// TIA Portal V16 export
// export: Created 2024-06-17T18:37:11.9513972Z, ExportSetting WithDefaults, DisplayName Totally Integrated Automation Portal, DisplayVersion V16, DisplayName TIA Portal Version Control Interface, DisplayVersion V16, DisplayName TIA Portal Openness, DisplayVersion V16, DisplayName STEP 7 Professional, DisplayVersion V16, DisplayName STEP 7 Safety, DisplayVersion V16, DisplayName WinCC Advanced, DisplayVersion V16
TYPE "Axis.RB.Do_PLC.Di"
TITLE = Tabela de Entradas vindas do robô
// stored: IsFailsafeCompliant false
   STRUCT
      "RB.Go_PLC.GiPLC_NumProg" : Int;   // Retorno Número Programa em Execução
      "RB.Do_PLC.Di16_ProgramaRecebido" : Bool;   // Reconhecimento de Programa Recebido
      "RB.Do_PLC.Di17_RequisicaoPrograma" : Bool;   // Autoriza CLP a enviar Número de Programa
      "RB.Do_PLC.Di18_Home" : Bool;   // Robô em Home
      "RB.Do_PLC.Di19_FaultSumSignal" : Bool;   // Robo em Falha
      "RB.Do_PLC.Di20_SafetyChainOK" : Bool;   // Sem Falhas de Hardware nos Canais de Segurança
      "RB.Do_PLC.Di21_MotorOnState" : Bool;   // Motores Ligados
      "RB.Do_PLC.Di22_Auto_On" : Bool;   // Robô em Automático
      "RB.Do_PLC.Di23_Cycle_On" : Bool;   // Programa em Execução
      "RB.Do_PLC.Di24_EmCicloVazio" : Bool;   // Retorno de Ciclo Vazio Ativo
      "RB.Do_PLC.Di25_CicloParado" : Bool;   // Robo Parado Autoriza Entrada na Célula
      "RB.Do_PLC.Di26_SupervisaoMovLigada" : Bool;   // Envia Status de supervisão de movimento ligada
      "RB.Do_PLC.Di27_ColisaoDetectada" : Bool;   // Envia Status de colisão detectada pela supervisão de movimento
      "RB.Do_PLC.Di28_EmPosManutencao" : Bool;   // Em Posição de Manutenção
      "RB.Do_PLC.Di29_EmPosCalibracao" : Bool;   // Em Posição de Calibração
      "RB.Do_PLC.Di30_EmPosSincronisco" : Bool;   // Em Posição de Sincronismo
      "RB.Do_PLC.Di31_Reserva" : Bool;   // Reserva
      "RB.Do_PLC.Di32_FalhaAr" : Bool;   // Status de falha de ar
      "RB.Do_PLC.Di33_FalhaAgua" : Bool;   // Status de falha de água
      "RB.Do_PLC.Di34_FalhaSolda" : Bool;   // Status de falha de solda
      "RB.Do_PLC.Di35_FalhaToolChanger" : Bool;   // Status de falha Tool Changer
      "RB.Do_PLC.Di36_FalhaPrograma" : Bool;   // Status de falha no programa do robô
      "RB.Do_PLC.Di37_FalhaFresagem" : Bool;   // Status de falha na execução da fresagem
      "RB.Do_PLC.Di38_Reserva" : Bool;   // Reserva
      "RB.Do_PLC.Di39_Reserva" : Bool;   // Reserva
      "RB.Do_PLC.Di40_Reserva" : Bool;   // Reserva
      "RB.Do_PLC.Di41_Reserva" : Bool;   // Reserva
      "RB.Do_PLC.Di42_Reserva" : Bool;   // Reserva
      "RB.Do_PLC.Di43_Reserva" : Bool;   // Reserva
      "RB.Do_PLC.Di44_Reserva" : Bool;   // Reserva
      "RB.Do_PLC.Di45_Reserva" : Bool;   // Reserva
      "RB.Do_PLC.Di46_Reserva" : Bool;   // Reserva
      "RB.Do_PLC.Di47_Reserva" : Bool;   // Reserva
      "RB.Do_PLC.Di48_Reserva" : Bool;   // Reserva
      "RB.Do_PLC.Di49_Reserva" : Bool;   // Reserva
      "RB.Do_PLC.Di50_Reserva" : Bool;   // Reserva
      "RB.Do_PLC.Di51_Reserva" : Bool;   // Reserva
      "RB.Do_PLC.Di52_Reserva" : Bool;   // Reserva
      "RB.Do_PLC.Di53_Reserva" : Bool;   // Reserva
      "RB.Do_PLC.Di54_Reserva" : Bool;   // Reserva
      "RB.Do_PLC.Di55_Reserva" : Bool;   // Reserva
      "RB.Do_PLC.Di56_AreaLivreTrab_1" : Bool;   // Robo Fora da Área de Trabalho 1
      "RB.Do_PLC.Di57_AreaLivreTrab_2" : Bool;   // Robo Fora da Área de Trabalho 2
      "RB.Do_PLC.Di58_AreaLivreTrab_3" : Bool;   // Robo Fora da Área de Trabalho 3
      "RB.Do_PLC.Di59_AreaLivreTrab_4" : Bool;   // Robo Fora da Área de Trabalho 4
      "RB.Do_PLC.Di60_AreaLivreTrab_5" : Bool;   // Robo Fora da Área de Trabalho 5
      "RB.Do_PLC.Di61_AreaLivreTrab_6" : Bool;   // Robo Fora da Área de Trabalho 6
      "RB.Do_PLC.Di62_AreaLivreTrab_7" : Bool;   // Robo Fora da Área de Trabalho 7
      "RB.Do_PLC.Di63_AreaLivreTrab_8" : Bool;   // Robo Fora da Área de Trabalho 8
      "RB.Do_PLC.Di64_AreaLivreTrab_9" : Bool;   // Robo Fora da Área de Trabalho 9
      "RB.Do_PLC.Di65_AreaLivreTrab_10" : Bool;   // Robo Fora da Área de Trabalho 10
      "RB.Do_PLC.Di66_AreaLivreTrab_11" : Bool;   // Robo Fora da Área de Trabalho 11
      "RB.Do_PLC.Di67_AreaLivreTrab_12" : Bool;   // Robo Fora da Área de Trabalho 12
      "RB.Do_PLC.Di68_AreaLivreTrab_13" : Bool;   // Robo Fora da Área de Trabalho 13
      "RB.Do_PLC.Di69_AreaLivreTrab_14" : Bool;   // Robo Fora da Área de Trabalho 14
      "RB.Do_PLC.Di70_AreaLivreTrab_15" : Bool;   // Robo Fora da Área de Trabalho 15
      "RB.Do_PLC.Di71_AreaLivreTrab_16" : Bool;   // Robo Fora da Área de Trabalho 16
      "RB.Do_PLC.Di72_AreaLivreTrab_17" : Bool;   // Robo Fora da Área de Trabalho 17
      "RB.Do_PLC.Di73_AreaLivreTrab_18" : Bool;   // Robo Fora da Área de Trabalho 18
      "RB.Do_PLC.Di74_AreaLivreTrab_19" : Bool;   // Robo Fora da Área de Trabalho 19
      "RB.Do_PLC.Di75_AreaLivreTrab_20" : Bool;   // Robo Fora da Área de Trabalho 20
      "RB.Do_PLC.Di76_AreaLivreTrab_21" : Bool;   // Robo Fora da Área de Trabalho 21
      "RB.Do_PLC.Di77_AreaLivreTrab_22" : Bool;   // Robo Fora da Área de Trabalho 22
      "RB.Do_PLC.Di78_AreaLivreTrab_23" : Bool;   // Robo Fora da Área de Trabalho 23
      "RB.Do_PLC.Di79_AreaLivreTrab_24" : Bool;   // Robo Fora da Área de Trabalho 24
      "RB.Do_PLC.Di80_AreaLivreTrab_25" : Bool;   // Robo Fora da Área de Trabalho 25
      "RB.Do_PLC.Di81_AreaLivreTrab_26" : Bool;   // Robo Fora da Área de Trabalho 26
      "RB.Do_PLC.Di82_AreaLivreTrab_27" : Bool;   // Robo Fora da Área de Trabalho 27
      "RB.Do_PLC.Di83_AreaLivreTrab_28" : Bool;   // Robo Fora da Área de Trabalho 28
      "RB.Do_PLC.Di84_AreaLivreTrab_29" : Bool;   // Robo Fora da Área de Trabalho 29
      "RB.Do_PLC.Di85_AreaLivreTrab_30" : Bool;   // Robo Fora da Área de Trabalho 30
      "RB.Do_PLC.Di86_AreaLivreTrab_31" : Bool;   // Robo Fora da Área de Trabalho 31
      "RB.Do_PLC.Di87_AreaLivreTrab_32" : Bool;   // Robo Fora da Área de Trabalho 32
      "RB.Do_PLC.Di88_Intertravamento_1" : Bool;   // Requisita Acesso Área de Intertravamento 1
      "RB.Do_PLC.Di89_Intertravamento_2" : Bool;   // Requisita Acesso Área de Intertravamento 2
      "RB.Do_PLC.Di90_Intertravamento_3" : Bool;   // Requisita Acesso Área de Intertravamento 3
      "RB.Do_PLC.Di91_Intertravamento_4" : Bool;   // Requisita Acesso Área de Intertravamento 4
      "RB.Do_PLC.Di92_Intertravamento_5" : Bool;   // Requisita Acesso Área de Intertravamento 5
      "RB.Do_PLC.Di93_Intertravamento_6" : Bool;   // Requisita Acesso Área de Intertravamento 6
      "RB.Do_PLC.Di94_Intertravamento_7" : Bool;   // Requisita Acesso Área de Intertravamento 7
      "RB.Do_PLC.Di95_Intertravamento_8" : Bool;   // Requisita Acesso Área de Intertravamento 8
      "RB.Do_PLC.Di96_Intertravamento_9" : Bool;   // Requisita Acesso Área de Intertravamento 9
      "RB.Do_PLC.Di97_Intertravamento_10" : Bool;   // Requisita Acesso Área de Intertravamento 10
      "RB.Do_PLC.Di98_Intertravamento_11" : Bool;   // Requisita Acesso Área de Intertravamento 11
      "RB.Do_PLC.Di99_Intertravamento_12" : Bool;   // Requisita Acesso Área de Intertravamento 12
      "RB.Do_PLC.Di100_Intertravamento_13" : Bool;   // Requisita Acesso Área de Intertravamento 13
      "RB.Do_PLC.Di101_Intertravamento_14" : Bool;   // Requisita Acesso Área de Intertravamento 14
      "RB.Do_PLC.Di102_Intertravamento_15" : Bool;   // Requisita Acesso Área de Intertravamento 15
      "RB.Do_PLC.Di103_Intertravamento_16" : Bool;   // Requisita Acesso Área de Intertravamento 16
      "RB.Do_PLC.Di104_Intertravamento_17" : Bool;   // Requisita Acesso Área de Intertravamento 17
      "RB.Do_PLC.Di105_Intertravamento_18" : Bool;   // Requisita Acesso Área de Intertravamento 18
      "RB.Do_PLC.Di106_Intertravamento_19" : Bool;   // Requisita Acesso Área de Intertravamento 19
      "RB.Do_PLC.Di107_Intertravamento_20" : Bool;   // Requisita Acesso Área de Intertravamento 20
      "RB.Do_PLC.Di108_Intertravamento_21" : Bool;   // Requisita Acesso Área de Intertravamento 21
      "RB.Do_PLC.Di109_Intertravamento_22" : Bool;   // Requisita Acesso Área de Intertravamento 22
      "RB.Do_PLC.Di110_Intertravamento_23" : Bool;   // Requisita Acesso Área de Intertravamento 23
      "RB.Do_PLC.Di111_Intertravamento_24" : Bool;   // Requisita Acesso Área de Intertravamento 24
      "RB.Do_PLC.Di112_Intertravamento_25" : Bool;   // Requisita Acesso Área de Intertravamento 25
      "RB.Do_PLC.Di113_Intertravamento_26" : Bool;   // Requisita Acesso Área de Intertravamento 26
      "RB.Do_PLC.Di114_Intertravamento_27" : Bool;   // Requisita Acesso Área de Intertravamento 27
      "RB.Do_PLC.Di115_Intertravamento_28" : Bool;   // Requisita Acesso Área de Intertravamento 28
      "RB.Do_PLC.Di116_Intertravamento_29" : Bool;   // Requisita Acesso Área de Intertravamento 29
      "RB.Do_PLC.Di117_Intertravamento_30" : Bool;   // Requisita Acesso Área de Intertravamento 30
      "RB.Do_PLC.Di118_Intertravamento_31" : Bool;   // Requisita Acesso Área de Intertravamento 31
      "RB.Do_PLC.Di119_Intertravamento_32" : Bool;   // Requisita Acesso Área de Intertravamento 32
      "RB.Do_PLC.Di120_FimTrabalho_1" : Bool;   // Fim de Trabalho 1
      "RB.Do_PLC.Di121_FimTrabalho_2" : Bool;   // Fim de Trabalho 2
      "RB.Do_PLC.Di122_FimTrabalho_3" : Bool;   // Fim de Trabalho 3
      "RB.Do_PLC.Di123_FimTrabalho_4" : Bool;   // Fim de Trabalho 4
      "RB.Do_PLC.Di124_FimTrabalho_5" : Bool;   // Fim de Trabalho 5
      "RB.Do_PLC.Di125_FimTrabalho_6" : Bool;   // Fim de Trabalho 6
      "RB.Do_PLC.Di126_FimTrabalho_7" : Bool;   // Fim de Trabalho 7
      "RB.Do_PLC.Di127_FimTrabalho_8" : Bool;   // Fim de Trabalho 8
      "RB.Do_PLC.Di128_FimTrabalho_9" : Bool;   // Fim de Trabalho 9
      "RB.Do_PLC.Di129_FimTrabalho_10" : Bool;   // Fim de Trabalho 10
      "RB.Do_PLC.Di130_FimTrabalho_11" : Bool;   // Fim de Trabalho 11
      "RB.Do_PLC.Di131_FimTrabalho_12" : Bool;   // Fim de Trabalho 12
      "RB.Do_PLC.Di132_FimTrabalho_13" : Bool;   // Fim de Trabalho 13
      "RB.Do_PLC.Di133_FimTrabalho_14" : Bool;   // Fim de Trabalho 14
      "RB.Do_PLC.Di134_FimTrabalho_15" : Bool;   // Fim de Trabalho 15
      "RB.Do_PLC.Di135_FimTrabalho_16" : Bool;   // Fim de Trabalho 16
      "RB.Do_PLC.Di136_FimTrabalho_17" : Bool;   // Fim de Trabalho 17
      "RB.Do_PLC.Di137_FimTrabalho_18" : Bool;   // Fim de Trabalho 18
      "RB.Do_PLC.Di138_FimTrabalho_19" : Bool;   // Fim de Trabalho 19
      "RB.Do_PLC.Di139_FimTrabalho_20" : Bool;   // Fim de Trabalho 20
      "RB.Do_PLC.Di140_FimTrabalho_21" : Bool;   // Fim de Trabalho 21
      "RB.Do_PLC.Di141_FimTrabalho_22" : Bool;   // Fim de Trabalho 22
      "RB.Do_PLC.Di142_FimTrabalho_23" : Bool;   // Fim de Trabalho 23
      "RB.Do_PLC.Di143_FimTrabalho_24" : Bool;   // Fim de Trabalho 24
      "RB.Do_PLC.Di144_FimTrabalho_25" : Bool;   // Fim de Trabalho 25
      "RB.Do_PLC.Di145_FimTrabalho_26" : Bool;   // Fim de Trabalho 26
      "RB.Do_PLC.Di146_FimTrabalho_27" : Bool;   // Fim de Trabalho 27
      "RB.Do_PLC.Di147_FimTrabalho_28" : Bool;   // Fim de Trabalho 28
      "RB.Do_PLC.Di148_FimTrabalho_29" : Bool;   // Fim de Trabalho 29
      "RB.Do_PLC.Di149_FimTrabalho_30" : Bool;   // Fim de Trabalho 30
      "RB.Do_PLC.Di150_FimTrabalho_31" : Bool;   // Fim de Trabalho 31
      "RB.Do_PLC.Di151_FimTrabalho_32" : Bool;   // Fim de Trabalho 32
      "RB.Do_PLC.Di152_NumEquip_B0" : Bool;   // Retorna Número do Equipamento Acoplado Bit 0
      "RB.Do_PLC.Di153_NumEquip_B1" : Bool;   // Retorna Número do Equipamento Acoplado Bit 1
      "RB.Do_PLC.Di154_NumEquip_B2" : Bool;   // Retorna Número do Equipamento Acoplado Bit 2
      "RB.Do_PLC.Di155_NumEquip_B3" : Bool;   // Retorna Número do Equipamento Acoplado Bit 3
      "RB.Do_PLC.Di156_NumEquip_B4" : Bool;   // Retorna Número do Equipamento Acoplado Bit 4
      "RB.Do_PLC.Di157_NumEquip_B5" : Bool;   // Retorna Número do Equipamento Acoplado Bit 5
      "RB.Do_PLC.Di158_NumEquip_B6" : Bool;   // Retorna Número do Equipamento Acoplado Bit 6
      "RB.Do_PLC.Di159_NumEquip_B7" : Bool;   // Retorna Número do Equipamento Acoplado Bit 7
      "RB.Do_PLC.Di160_ReqAtivarPnetEquip_1" : Bool;   // Requisição Ativar Rede Profinet Equipamento 1
      "RB.Do_PLC.Di161_ReqAtivarPnetEquip_2" : Bool;   // Requisição Ativar Rede Profinet Equipamento 2
      "RB.Do_PLC.Di162_ReqAtivarPnetEquip_3" : Bool;   // Requisição Ativar Rede Profinet Equipamento 3
      "RB.Do_PLC.Di163_ReqAtivarPnetEquip_4" : Bool;   // Requisição Ativar Rede Profinet Equipamento 4
      "RB.Do_PLC.Di164_ReqAtivarPnetEquip_5" : Bool;   // Requisição Ativar Rede Profinet Equipamento 5
      "RB.Do_PLC.Di165_ReqAtivarPnetEquip_6" : Bool;   // Requisição Ativar Rede Profinet Equipamento 6
      "RB.Do_PLC.Di166_ReqAtivarPnetEquip_7" : Bool;   // Requisição Ativar Rede Profinet Equipamento 7
      "RB.Do_PLC.Di167_ReqAtivarPnetEquip_8" : Bool;   // Requisição Ativar Rede Profinet Equipamento 8
      "RB.Do_PLC.Di168_ReqDesatPnetEquip_1" : Bool;   // Requisição Desativar Rede Profinet Equipamento 1
      "RB.Do_PLC.Di169_ReqDesatPnetEquip_2" : Bool;   // Requisição Desativar Rede Profinet Equipamento 2
      "RB.Do_PLC.Di170_ReqDesatPnetEquip_3" : Bool;   // Requisição Desativar Rede Profinet Equipamento 3
      "RB.Do_PLC.Di171_ReqDesatPnetEquip_4" : Bool;   // Requisição Desativar Rede Profinet Equipamento 4
      "RB.Do_PLC.Di172_ReqDesatPnetEquip_5" : Bool;   // Requisição Desativar Rede Profinet Equipamento 5
      "RB.Do_PLC.Di173_ReqDesatPnetEquip_6" : Bool;   // Requisição Desativar Rede Profinet Equipamento 6
      "RB.Do_PLC.Di174_ReqDesatPnetEquip_7" : Bool;   // Requisição Desativar Rede Profinet Equipamento 7
      "RB.Do_PLC.Di175_ReqDesatPnetEquip_8" : Bool;   // Requisição Desativar Rede Profinet Equipamento 8
      "RB.Do_PLC.Di176_EmPosTrEletEquip_1" : Bool;   // Em Posição de Troca de Eletrodo Equipamento 1
      "RB.Do_PLC.Di177_EmPosTrEletEquip_2" : Bool;   // Em Posição de Troca de Eletrodo Equipamento 2
      "RB.Do_PLC.Di178_EmPosTrEletEquip_3" : Bool;   // Em Posição de Troca de Eletrodo Equipamento 3
      "RB.Do_PLC.Di179_EmPosTrEletEquip_4" : Bool;   // Em Posição de Troca de Eletrodo Equipamento 4
      "RB.Do_PLC.Di180_EmPosTrEletEquip_5" : Bool;   // Em Posição de Troca de Eletrodo Equipamento 5
      "RB.Do_PLC.Di181_EmPosTrEletEquip_6" : Bool;   // Em Posição de Troca de Eletrodo Equipamento 6
      "RB.Do_PLC.Di182_EmPosTrEletEquip_7" : Bool;   // Em Posição de Troca de Eletrodo Equipamento 7
      "RB.Do_PLC.Di183_EmPosTrEletEquip_8" : Bool;   // Em Posição de Troca de Eletrodo Equipamento 8
      "RB.Do_PLC.Di184_FresaEfetuadaEquip_1" : Bool;   // Fresa Efetuada Equipamento 1
      "RB.Do_PLC.Di185_FresaEfetuadaEquip_2" : Bool;   // Fresa Efetuada Equipamento 2
      "RB.Do_PLC.Di186_FresaEfetuadaEquip_3" : Bool;   // Fresa Efetuada Equipamento 3
      "RB.Do_PLC.Di187_FresaEfetuadaEquip_4" : Bool;   // Fresa Efetuada Equipamento 4
      "RB.Do_PLC.Di188_FresaEfetuadaEquip_5" : Bool;   // Fresa Efetuada Equipamento 5
      "RB.Do_PLC.Di189_FresaEfetuadaEquip_6" : Bool;   // Fresa Efetuada Equipamento 6
      "RB.Do_PLC.Di190_FresaEfetuadaEquip_7" : Bool;   // Fresa Efetuada Equipamento 7
      "RB.Do_PLC.Di191_FresaEfetuadaEquip_8" : Bool;   // Fresa Efetuada Equipamento 8
      "RB.Do_PLC.Di192_AvisoTrEletEquip_1" : Bool;   // Aviso (Pré-Alarme) Troca de Eletrodo Equipamento 1
      "RB.Do_PLC.Di193_AvisoTrEletEquip_2" : Bool;   // Aviso (Pré-Alarme) Troca de Eletrodo Equipamento 2
      "RB.Do_PLC.Di194_AvisoTrEletEquip_3" : Bool;   // Aviso (Pré-Alarme) Troca de Eletrodo Equipamento 3
      "RB.Do_PLC.Di195_AvisoTrEletEquip_4" : Bool;   // Aviso (Pré-Alarme) Troca de Eletrodo Equipamento 4
      "RB.Do_PLC.Di196_AvisoTrEletEquip_5" : Bool;   // Aviso (Pré-Alarme) Troca de Eletrodo Equipamento 5
      "RB.Do_PLC.Di197_AvisoTrEletEquip_6" : Bool;   // Aviso (Pré-Alarme) Troca de Eletrodo Equipamento 6
      "RB.Do_PLC.Di198_AvisoTrEletEquip_7" : Bool;   // Aviso (Pré-Alarme) Troca de Eletrodo Equipamento 7
      "RB.Do_PLC.Di199_AvisoTrEletEquip_8" : Bool;   // Aviso (Pré-Alarme) Troca de Eletrodo Equipamento 8
      "RB.Do_PLC.Di200_AlarmeTrEletEquip_1" : Bool;   // Alarme Troca de Eletrodo Equipamento 1
      "RB.Do_PLC.Di201_AlarmeTrEletEquip_2" : Bool;   // Alarme Troca de Eletrodo Equipamento 2
      "RB.Do_PLC.Di202_AlarmeTrEletEquip_3" : Bool;   // Alarme Troca de Eletrodo Equipamento 3
      "RB.Do_PLC.Di203_AlarmeTrEletEquip_4" : Bool;   // Alarme Troca de Eletrodo Equipamento 4
      "RB.Do_PLC.Di204_AlarmeTrEletEquip_5" : Bool;   // Alarme Troca de Eletrodo Equipamento 5
      "RB.Do_PLC.Di205_AlarmeTrEletEquip_6" : Bool;   // Alarme Troca de Eletrodo Equipamento 6
      "RB.Do_PLC.Di206_AlarmeTrEletEquip_7" : Bool;   // Alarme Troca de Eletrodo Equipamento 7
      "RB.Do_PLC.Di207_AlarmeTrEletEquip_8" : Bool;   // Alarme Troca de Eletrodo Equipamento 8
      "RB.Do_PLC.Di208_FuncaoAtivaEquip_1" : Bool;   // Retorna Informação que a Função Está Ativa Equipamento 1
      "RB.Do_PLC.Di209_FuncaoAtivaEquip_2" : Bool;   // Retorna Informação que a Função Está Ativa Equipamento 2
      "RB.Do_PLC.Di210_FuncaoAtivaEquip_3" : Bool;   // Retorna Informação que a Função Está Ativa Equipamento 3
      "RB.Do_PLC.Di211_FuncaoAtivaEquip_4" : Bool;   // Retorna Informação que a Função Está Ativa Equipamento 4
      "RB.Do_PLC.Di212_FuncaoAtivaEquip_5" : Bool;   // Retorna Informação que a Função Está Ativa Equipamento 5
      "RB.Do_PLC.Di213_FuncaoAtivaEquip_6" : Bool;   // Retorna Informação que a Função Está Ativa Equipamento 6
      "RB.Do_PLC.Di214_FuncaoAtivaEquip_7" : Bool;   // Retorna Informação que a Função Está Ativa Equipamento 7
      "RB.Do_PLC.Di215_FuncaoAtivaEquip_8" : Bool;   // Retorna Informação que a Função Está Ativa Equipamento 8
      "RB.Do_PLC.Di216_Req.Ava_Grupo_A" : Bool;   // Requisição de Avanço Grupo A
      "RB.Do_PLC.Di217_Req.Ava_Grupo_B" : Bool;   // Requisição de Avanço Grupo B
      "RB.Do_PLC.Di218_Req.Ava_Grupo_C" : Bool;   // Requisição de Avanço Grupo C
      "RB.Do_PLC.Di219_Req.Ava_Grupo_D" : Bool;   // Requisição de Avanço Grupo D
      "RB.Do_PLC.Di220_Req.Ava_Grupo_E" : Bool;   // Requisição de Avanço Grupo E
      "RB.Do_PLC.Di221_Req.Ava_Grupo_F" : Bool;   // Requisição de Avanço Grupo F
      "RB.Do_PLC.Di222_Req.Ava_Grupo_G" : Bool;   // Requisição de Avanço Grupo G
      "RB.Do_PLC.Di223_Req.Ava_Grupo_H" : Bool;   // Requisição de Avanço Grupo H
      "RB.Do_PLC.Di224_Req.Ava_Grupo_I" : Bool;   // Requisição de Avanço Grupo I
      "RB.Do_PLC.Di225_Req.Ava_Grupo_J" : Bool;   // Requisição de Avanço Grupo J
      "RB.Do_PLC.Di226_Req.Ava_Grupo_K" : Bool;   // Requisição de Avanço Grupo K
      "RB.Do_PLC.Di227_Req.Ava_Grupo_L" : Bool;   // Requisição de Avanço Grupo L
      "RB.Do_PLC.Di228_Req.Ava_Grupo_M" : Bool;   // Requisição de Avanço Grupo M
      "RB.Do_PLC.Di229_Req.Ava_Grupo_N" : Bool;   // Requisição de Avanço Grupo N
      "RB.Do_PLC.Di230_Req.Ava_Grupo_O" : Bool;   // Requisição de Avanço Grupo O
      "RB.Do_PLC.Di231_Req.Ava_Grupo_P" : Bool;   // Requisição de Avanço Grupo P
      "RB.Do_PLC.Di232_Req.Rec_Grupo_A" : Bool;   // Requisição de Recuo Grupo A
      "RB.Do_PLC.Di233_Req.Rec_Grupo_B" : Bool;   // Requisição de Recuo Grupo B
      "RB.Do_PLC.Di234_Req.Rec_Grupo_C" : Bool;   // Requisição de Recuo Grupo C
      "RB.Do_PLC.Di235_Req.Rec_Grupo_D" : Bool;   // Requisição de Recuo Grupo D
      "RB.Do_PLC.Di236_Req.Rec_Grupo_E" : Bool;   // Requisição de Recuo Grupo E
      "RB.Do_PLC.Di237_Req.Rec_Grupo_F" : Bool;   // Requisição de Recuo Grupo F
      "RB.Do_PLC.Di238_Req.Rec_Grupo_G" : Bool;   // Requisição de Recuo Grupo G
      "RB.Do_PLC.Di239_Req.Rec_Grupo_H" : Bool;   // Requisição de Recuo Grupo H
      "RB.Do_PLC.Di240_Req.Rec_Grupo_I" : Bool;   // Requisição de Recuo Grupo I
      "RB.Do_PLC.Di241_Req.Rec_Grupo_J" : Bool;   // Requisição de Recuo Grupo J
      "RB.Do_PLC.Di242_Req.Rec_Grupo_K" : Bool;   // Requisição de Recuo Grupo K
      "RB.Do_PLC.Di243_Req.Rec_Grupo_L" : Bool;   // Requisição de Recuo Grupo L
      "RB.Do_PLC.Di244_Req.Rec_Grupo_M" : Bool;   // Requisição de Recuo Grupo M
      "RB.Do_PLC.Di245_Req.Rec_Grupo_N" : Bool;   // Requisição de Recuo Grupo N
      "RB.Do_PLC.Di246_Req.Rec_Grupo_O" : Bool;   // Requisição de Recuo Grupo O
      "RB.Do_PLC.Di247_Req.Rec_Grupo_P" : Bool;   // Requisição de Recuo Grupo P
      "RB.Do_PLC.Di248_ReqMovimentoDisp_1" : Bool;   // Dispositivo: Requisição Movimento 1
      "RB.Do_PLC.Di249_ReqMovimentoDisp_2" : Bool;   // Dispositivo: Requisição Movimento 2
      "RB.Do_PLC.Di250_ReqMovimentoDisp_3" : Bool;   // Dispositivo: Requisição Movimento 3
      "RB.Do_PLC.Di251_ReqMovimentoDisp_4" : Bool;   // Dispositivo: Requisição Movimento 4
      "RB.Do_PLC.Di252_ReqMovimentoDisp_5" : Bool;   // Dispositivo: Requisição Movimento 5
      "RB.Do_PLC.Di253_ReqMovimentoDisp_6" : Bool;   // Dispositivo: Requisição Movimento 6
      "RB.Do_PLC.Di254_ReqMovimentoDisp_7" : Bool;   // Dispositivo: Requisição Movimento 7
      "RB.Do_PLC.Di255_ReqMovimentoDisp_8" : Bool;   // Dispositivo: Requisição Movimento 8
   END_STRUCT;
END_TYPE
